FUNCTION_BLOCK ARUCODETECTOR (* openCV Aruco Detector *)
  (* Version 1.0, AN, SWDC RTSoft *)
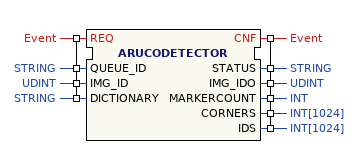
  EVENT_INPUT
    REQ WITH QUEUE_ID, IMG_ID, DICTIONARY;
  END_EVENT
  EVENT_OUTPUT
    CNF WITH STATUS, IMG_IDO, MARKERCOUNT, CORNERS, IDS;
  END_EVENT
  VAR_INPUT
    QUEUE_ID : STRING;
    IMG_ID : UDINT;
    DICTIONARY : STRING; (* Dictionary format: 4X4_50, 6x6_250, 6*6_250. Case insensitive *)
  END_VAR
  VAR_OUTPUT
    STATUS : STRING;
    IMG_IDO : UDINT;
    MARKERCOUNT : INT; (* Number of detected Aruco markers *)
    CORNERS : ARRAY [0..1023] OF INT; (* Detected Aruco marker corners *)
    IDS : ARRAY [0..1023] OF INT; (* Detected Aruco marker IDs *)
  END_VAR
  ALGORITHM REQ IN ST:

  END_ALGORITHM
END_FUNCTION_BLOCK
